{attribute 'conditionalshow'}
FUNCTION_BLOCK FB_CV_WORD_TO_UDINT
VAR_INPUT
	{attribute 'hide'}
	wInputValue_1				: WORD;								//Input value that is converted into the output value
	{attribute 'hide'}
	wInputValue_2				: WORD;								//Input value that is converted into the output value
	{attribute 'hide'}
	eByteOrderForConvert		: eByteOrder;						//Byte Format
END_VAR
VAR_OUTPUT
	{attribute 'hide'}
	udiOutputValue				: UDINT;							//Converted output value							
END_VAR
VAR
END_VAR

//Creator : Kai Ebensperger
//Company : Lynus AG
//Date : 28.04.2021
//Version : 1.0.0.0

//With this functionblock its possible to convert a certain Datatyp in a other Datatype
//The byte order can be selected between BigEndian and LittleEndian
//WORD TO UDINT
//Created for the Edge Device Lib over Modbus TCP
//Modbus TCP is WORD oriented

IF eByteOrderForConvert = eByteOrder.eBigEndian THEN
	udiOutputValue := SHL(WORD_TO_UDINT(wInputValue_1),16) + WORD_TO_UDINT(wInputValue_2);
ELSE
	udiOutputValue := SHL(WORD_TO_UDINT(wInputValue_2),16) + WORD_TO_UDINT(wInputValue_1);
END_IF

END_FUNCTION_BLOCK

(* stored: Version 1.1.0.1, ProductVersion 3.1.4024.9
   POU FB_CV_WORD_TO_UDINT: Id {3ff5f54d-6c59-4568-a537-efae3b29a6d8}, SpecialFunc None *)
